{attribute 'enable_dynamic_creation'}
FUNCTION_BLOCK FB_Motor IMPLEMENTS I_Object
VAR_INPUT
END_VAR
VAR_OUTPUT
END_VAR
VAR
	sObjectID			: STRING;
	eObjectType			: E_OBJECTS;
	// pointers for destructor
	_pInstance			: POINTER TO FB_Motor;
	_pTemp				: POINTER TO FB_Motor;
END_VAR

METHOD Destruct : BOOL
// destroy the instance 
IF _pInstance	<> 0 THEN
	// store in temp value otherwise the FB_exit called at __DELETE will create a stack overflow
	// when not set to 0 before __DELETE  
	_pTemp := _pInstance;
	_pInstance := 16#0; 
	__DELETE(_pTemp);
END_IF
END_METHOD

METHOD FB_init : BOOL
VAR_INPUT
	bInitRetains       : BOOL; // if TRUE, the retain variables are initialized (warm start / cold start)
	bInCopyCode        : BOOL;  // if TRUE, the instance afterwards gets moved into the copy code (online change)
	// Object identifier name
	sObjectID			: STRING;	
	// Object type as a string
	eObjectType			: E_OBJECTS;
END_VAR
THIS^.sObjectID		:= sObjectID;
THIS^.eObjectType	:= eObjectType;
END_METHOD

METHOD M_GetObjectDescription : string
VAR_INPUT
END_VAR
VAR
	sDescription			: STRING;
END_VAR
sDescription := concat(THIS^.sObjectID, ' Type: '); 
sDescription := concat(sDescription, TO_STRING(THIS^.eObjectType)); 
M_GetObjectDescription := sDescription;
END_METHOD

{warning 'add method implementation'}
METHOD M_Reset : BOOL
END_METHOD

{warning 'add method implementation'}
METHOD M_Start : BOOL
END_METHOD

{warning 'add property implementation'}
PROPERTY P_Status : DWORD
GET
END_GET
END_PROPERTY

PROPERTY pInstance : POINTER TO FB_EmptyObject
SET
// Store pointer for destructor
_pInstance := pInstance;
END_SET
END_PROPERTY

END_FUNCTION_BLOCK

(* stored: Version 1.1.0.1, ProductVersion 3.1.4022.18
   POU FB_Motor: Id {16b3c71e-287b-4d59-8d9f-5bc2e78f4f25}, SpecialFunc None
   Method Destruct: Id {ecd132b5-e36b-4934-ab5a-54c517ae1042}
   Method FB_init: Id {d71bf903-5eee-4127-af9b-086d5281fe99}
   Method M_GetObjectDescription: Id {cc3e7c16-38bf-452b-a10b-5f9245753805}
   Method M_Reset: Id {8d0a7951-5ca1-41e0-bfb1-8acbad57749f}
   Method M_Start: Id {abfef9a7-d3ba-4cc9-b65b-9c5e2f44c5e9}
   Property P_Status: Id {0f503500-5690-4122-a899-5aa257fc48d9}
   Get Get: Id {47b53e07-f8c9-45b2-bd9a-65821a5dfee4}
   Property pInstance: Id {b495c143-1c4f-44f3-84ed-ccd96d6a5ffc}
   Set Set: Id {0aee5ea9-193d-4678-a451-6df8650e98e4} *)
